# EPICS autosave request: iocBoot/ioc13bmd_TOMO_XPS/auto_settings.req
file "CARS_motor_settings.req",         P=$(P), M=m121
file "CARS_motor_settings.req",         P=$(P), M=m122
file "CARS_motor_settings.req",         P=$(P), M=m123
file "CARS_motor_settings.req",         P=$(P), M=m124
#file "CARS_motor_settings.req",         P=$(P), M=m125
#file "CARS_motor_settings.req",         P=$(P), M=m126
#file "CARS_motor_settings.req",         P=$(P), M=m127
#file "CARS_motor_settings.req",         P=$(P), M=m128
